{attribute addProperty BoxType "KL1512"}
{attribute addProperty Id "Channel_1Channel_585D17BE00Channel_2Channel_585D17BE00"}
{attribute addProperty CRC "3457887495"}
{attribute addProperty SizeInBites "0"}
{attribute addProperty SizeInBytes "0"}
TYPE KL1512_CE1B2D07 :
STRUCT
	{attribute addProperty Name "Channel_1"}
	Channel_1 : Channel_585D17BE;
	{attribute addProperty Name "Channel_2"}
	Channel_2 : Channel_585D17BE;
END_STRUCT
END_TYPE

(* stored: Version 1.2.0.0, ProductVersion 3.1.4024.9
   DUT KL1512_CE1B2D07: Id {03fff6a9-09fd-4c7c-8d5d-245e1e6ae727} *)
